FUNCTION_BLOCK AR_CLIENT_1_0_EACH_EVENT (* Send a REAL from an AR adapter as a remote OPC-UA write via CLIENT_1_0 on EVERY IN.E1 trigger, unconditionally (no E_D_FF_ANY change-filter, unlike AR_CLIENT_1_0) *)
  (* Standard: 61499-2; Description: Copyright (c) 2026 HR Agrartechnik GmbH This program and the accompanying materials are made available under the terms of the Eclipse Public License 2.0 which is available at https://www.eclipse.org/legal/epl-2.0/ SPDX-License-Identifier: EPL-2.0 *)
  (* Version 1.0, 2026-09-25, Franz Höpfinger, HR Agrartechnik GmbH, initial implementation - AR_CLIENT_1_0-Variante OHNE E_D_FF_ANY-Value-Filter, fuer CALL_METHOD-Aufrufer, die JEDES echte Trigger-Event senden muessen, unabhaengig davon ob sich der Wert seit dem letzten Senden geaendert hat (bestaetigter Review-Fund auf PR #267: NumericValue_TO_CLIENT_1_0_OPC.SUB nutzte bisher AR_CLIENT_1_0, dessen interner E_D_FF_ANY einen erneuten VT/Web-Commit desselben Werts stillschweigend verschluckt - der eingegebene Wert war schon der zuletzt gesendete, die CALL_METHOD blieb aus. Hier entfaellt der Filter: IN.E1 loest F_MOVE/CLIENT_1_0.REQ direkt und immer aus. Bewusst als eigener Typ (nicht AR_CLIENT_1_0 selbst geaendert), weil AR_CLIENT_1_0's Change-Filter fuer andere, kuenftige Send-on-Change-Aufrufer weiterhin richtig/gewuenscht ist. *)
  PACKAGE adapter::net;
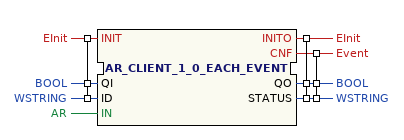
  EVENT_INPUT
    INIT : EInit WITH QI, ID; (* Initialization *)
  END_EVENT
  EVENT_OUTPUT
    INITO : EInit WITH QO, STATUS; (* Initialization Confirm *)
    CNF WITH QO, STATUS; (* Data was sent *)
  END_EVENT
  VAR_INPUT
    QI : BOOL;
    ID : WSTRING;
  END_VAR
  VAR_OUTPUT
    QO : BOOL;
    STATUS : WSTRING;
  END_VAR
  SOCKETS
    IN : adapter::types::unidirectional::AR; (* REAL to send, on every IN.E1 event *)
  END_SOCKETS
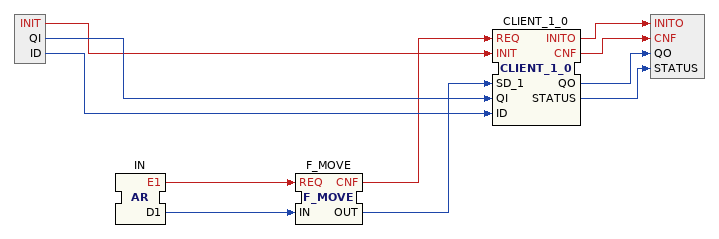
  FBS
    F_MOVE : iec61131::selection::F_MOVE; {SET_ATTRIBUTE(DataType, REAL)}
    CLIENT_1_0 : iec61499::net::CLIENT_1_0;
  END_FBS
  EVENT_CONNECTIONS
    CLIENT_1_0.INITO TO INITO;
    CLIENT_1_0.CNF TO CNF;
    IN.E1 TO F_MOVE.REQ;
    F_MOVE.CNF TO CLIENT_1_0.REQ;
    INIT TO CLIENT_1_0.INIT;
  END_CONNECTIONS
  DATA_CONNECTIONS
    CLIENT_1_0.QO TO QO;
    CLIENT_1_0.STATUS TO STATUS;
    IN.D1 TO F_MOVE.IN;
    F_MOVE.OUT TO CLIENT_1_0.SD_1;
    QI TO CLIENT_1_0.QI;
    ID TO CLIENT_1_0.ID;
  END_CONNECTIONS
END_FUNCTION_BLOCK
